FUNCTION_BLOCK FB_Task
VAR_INPUT
	iTaskNumber:USINT; //number of the task in the station, e.g. 1,2,3,4
	iEnableTask:BOOL; //TRUE to enable the task
	iBypassTask:BOOL; //TRUE to skip the task if not required for a particular complexity
	iStartTask:BOOL; //TRUE to start task
	iCompleteTask:BOOL; //TRUE if the task is complete
	iTaskName:STRING(255); //name of task
END_VAR
VAR_OUTPUT
	qComplexity:UINT; //complexity of task
END_VAR
VAR
	startosr:R_TRIG; //start osr
	endosr:R_TRIG; //end osr
	TaskRunning: BOOL;
	
	//task state OSRs
	osrNotStarted:R_TRIG;
	osrStarted:R_TRIG;
	osrCompleted:R_TRIG;
	osrPassed:R_TRIG;
	osrFailed:R_TRIG; //failed to perform process
	osrRejected:R_TRIG; //failed on guage test
	osrSkipped:R_TRIG;
	osrBypassed:R_TRIG;
	osrUnknown:R_TRIG;
	
END_VAR
VAR_IN_OUT
	iqPartData:typeStation; //insert station data
END_VAR









//theme:2mcGhpbWlyg

startosr(CLK:=iStartTask);
endosr(CLK:=iCompleteTask);

//call assign states
actAssignState();

//set base colour
iqPartData.part.tasks[iTaskNumber].StateColour := HMIColour.colourGreyBackground;

//set task name
iqPartData.part.tasks[iTaskNumber].singleTaskName := iTaskName;

IF iEnableTask THEN
	iqPartData.part.tasks[iTaskNumber].IsTaskEnabled := TRUE;
	ELSE
	iqPartData.part.tasks[iTaskNumber].IsTaskEnabled := FALSE;
END_IF

//start task
IF startosr.Q THEN
	TaskRunning:=TRUE; //start task
END_IF

//end task conditions
IF endosr.Q THEN
	TaskRunning:=FALSE;
	iqPartData.part.tasks[iTaskNumber].TaskStatus := TaskState.Completed;
END_IF

//increment task time
IF TaskRunning AND System.PulseHundredMilliSecond THEN
	iqPartData.part.tasks[iTaskNumber].TaskStatus := TaskState.Started;
	iqPartData.part.tasks[iTaskNumber].CycleTimeActual := iqPartData.part.tasks[iTaskNumber].CycleTimeActual + 0.1;
END_IF

IF iBypassTask THEN
	;
END_IF


//set colour based on pass/fail
IF  iqPartData.part.tasks[iTaskNumber].IsTaskPassed THEN //set outcome colour
	iqPartData.part.tasks[iTaskNumber].StateColour := HMIColour.colourGreen;
END_IF

IF  iqPartData.part.tasks[iTaskNumber].IsTaskFailed THEN //set outcome colour
	iqPartData.part.tasks[iTaskNumber].StateColour := HMIColour.colourRed;
END_IF


//sum of pass / fail = Task Complete
IF 	(iqPartData.part.tasks[iTaskNumber].IsTaskPassed OR
	iqPartData.part.tasks[iTaskNumber].IsTaskFailed) OR
	iqPartData.part.tasks[iTaskNumber].TaskStatus = TaskState.Bypassed THEN
	iqPartData.part.tasks[iTaskNumber].IsTaskComplete := TRUE;
	ELSE
	iqPartData.part.tasks[iTaskNumber].IsTaskComplete := FALSE;
END_IF


//move complexity to output
qComplexity := iqPartData.part.tasks[iTaskNumber].complexity;

ACTION actAssignState:
//OSR check for setting feedback
osrNotStarted		(CLK:=NOT iqPartData.part.PartPresent					);
osrStarted			(CLK:=iStartTask										);
osrCompleted		(CLK:=iCompleteTask										);
osrPassed			(CLK:=iqPartData.part.tasks[iTaskNumber].IsTaskPassed	);
osrFailed			(CLK:=iqPartData.part.tasks[iTaskNumber].IsTaskFailed	); //failed to perform process
osrRejected			(CLK:=iqPartData.part.tasks[iTaskNumber].IsTaskRejected	); //failed on guage test
osrSkipped			(CLK:=iqPartData.part.tasks[iTaskNumber].IsTaskSkipped	);
osrBypassed			(CLK:=iqPartData.part.tasks[iTaskNumber].IsTaskBypassed	);
osrUnknown			(CLK:=NOT iqPartData.part.PartPresent AND iqPartData.part.DataReadNOK	);

IF osrNotStarted.Q	THEN ;		ELSE	;		END_IF;
IF osrStarted.Q		THEN ;		ELSE	;		END_IF;
IF osrCompleted.Q	THEN ;		ELSE	;		END_IF;
IF osrPassed.Q		THEN ;		ELSE	;		END_IF;
IF osrFailed.Q		THEN ;		ELSE	;		END_IF;
IF osrRejected.Q	THEN ;		ELSE	;		END_IF;
IF osrSkipped.Q		THEN ;		ELSE	;		END_IF;
IF osrBypassed.Q	THEN ;		ELSE	;		END_IF;
IF osrUnknown.Q		THEN ;		ELSE	;		END_IF;
IF osrRejected.Q	THEN ;		ELSE	;		END_IF;
END_ACTION

END_FUNCTION_BLOCK

(* stored: Version 1.1.0.1, ProductVersion 3.1.4024.12
   POU FB_Task: Id {15173ef1-ba55-44a8-a63e-6bf619f6f525}, SpecialFunc None
   Action actAssignState: Id {37109fc0-0d72-408a-be10-beb38c4b6abe} *)
